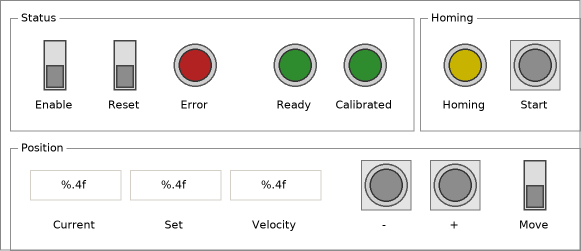
VISUALIZATION Azimuth  // 581x251
    GroupBox (10,10 404x121), "Status"
        DipSwitch (20,30 50x50), variable: MAIN.AzimuthControl.bEnable, behaviour: TOGGLE, style: Switch-DipSwitch-Gray
        DipSwitch (90,30 50x50), variable: MAIN.AzimuthControl.bReset, behaviour: TOGGLE, style: Switch-DipSwitch-Gray
        Lamp1 (160,30 50x50), variable: MAIN.AzimuthControl.bError, style: Lamp-Lamp1-Red
        Lamp1 (260,30 50x50), variable: MAIN.AzimuthControl.bReady, style: Lamp-Lamp1-Green
        Lamp1 (330,30 50x50), variable: MAIN.AzimuthControl.bCalibrated, style: Lamp-Lamp1-Green
        Label (10,80 68x30), "Enable"
        Label (80,80 68x30), "Reset"
        Label (150,80 68x30), "Error"
        Label (250,80 68x30), "Ready"
        Label (320,80 68x30), "Calibrated"
    GroupBox (420,10 161x121), "Homing"
        Lamp1 (20,30 50x50), variable: MAIN.AzimuthControl.bHomeAxis, style: Lamp-Lamp1-Yellow
        Label (10,80 68x30), "Homing"
        PushSwitch (90,30 50x50), variable: MAIN.AzimuthControl.bHomeAxis, behaviour: TOGGLE, style: Switch-PushSwitch-Gray
        Label (80,80 68x30), "Start"
    GroupBox (10,140 571x111), "Position"
        Textfield (20,30 91x30), "%.4f", text variable: MAIN.AzimuthControl.fActualPosition
        Label (30,70 68x30), "Current"
        Textfield (120,30 91x30), "%.4f", text variable: MAIN.AzimuthControl.fPosition
            OnMouseUp: write the text variable via InputWithLimits, min MAIN.AzimuthControl.fMinPosition, max MAIN.AzimuthControl.fMaxPosition
        Textfield (220,30 91x30), "%.4f", text variable: MAIN.AzimuthControl.fVelocity
            OnMouseUp: write the text variable via InputWithLimits, min 0, max 200
        PushSwitch (351,20 50x50), variable: MAIN.AzimuthControl.bMoveNeg, behaviour: TOGGLE, style: Switch-PushSwitch-Gray
        PushSwitch (420,20 50x50), variable: MAIN.AzimuthControl.bMovePos, behaviour: TOGGLE, style: Switch-PushSwitch-Gray
        DipSwitch (500,20 50x50), variable: MAIN.AzimuthControl.bMoveAxis, behaviour: TOGGLE, style: Switch-DipSwitch-Gray
        Label (340,70 68x30), "-"
        Label (410,70 68x30), "+"
        Label (490,70 68x30), "Move"
    Label (140,210 68x30), "Set"
    Label (240,210 68x30), "Velocity"
END_VISUALIZATION

(* stored: Version 1.1.0.1, ProductVersion 3.1.4024.15
   Visu Azimuth: Id {632e0126-0c13-4fd7-bb12-d5c69bed56cb} *)
